// TIA Portal V18 export
DATA_BLOCK "idbSpeedControl"   // DB1
// stored: InstanceOfName nsPerceuse.fbSpeedControl, InstanceOfType FB, Namespace nsPerceuse
"nsPerceuse.fbSpeedControl"
   // VAR_INPUT
   //    iFaster : Bool;
   //    iSlower : Bool;
   // END_VAR
   // VAR_IN_OUT
   //    ioSpeed : UDInt;
   // END_VAR
BEGIN
END_DATA_BLOCK
